(* Logix 5000 project; controller cal1615 1756-L62 rev 20.19; software revision 20.05; part 12 of 82 *)
(* tags used below, declared in another part *)
   tmrFlash : TIMER[4];   // Flash Timer
   aaa_aaa_temp : BOOL;
   FAULT : BOOL;   // Fault AFI
   FlashBit_500MSec : BOOL;   // Flash Bit 500 MSec
   HMI : BOOL;   // AFI HMI
   p00_FlashBit_1Sec : BOOL;   // System Flash Bit 1 Second
   p00_wac : Accumulator;   // Winder Accumulator
   p01_int_from_oxidizer : INT[10];   // System Oxidizer Int from Oxidizer
   p01_param_master_accel : REAL;   // Machine Parameter Master Accel Rate
   p01_param_master_decel : REAL;   // Machine Parameter Master Decel Rate
   p01_param_master_jog_accel : REAL;   // Machine Parameter Master Jog Acceleration mmpm/s
   p01_param_master_jog_decel : REAL;   // Machine Parameter Master Jog Deceleration mmpm/s
   p01_param_master_jog_speed : REAL;   // Machine Parameter Master Jog Speed
   p01_param_oven_timer_presets : DINT[32];   // System Parameter Oven Timer Presets
   p01_param_slow_speed_sp : REAL;   // System Parameters Slow Speed Setpoint
   p01_param_start_delay : REAL;   // Machine Parameter Start Delay
   p01_recipe_active : recipe;   // Active Recipe
   p01r01 : routine;
   p01r02_do_buzzer : BOOL;   // System Outputs Buzzer
   p01r02_do_horn : BOOL;   // System Outputs Horn
   p01r02_do_red_stack_light : BOOL;   // System Outputs Red Stack Light
   p01r02_do_yellow_stack_light : BOOL;   // System Outputs Yellow Stack Light
   p01r02_plc_scan_time_in_sec : REAL;   // System PLC Scan Time in Seconds
   p01r02_timer_second : TIMER[2];   // System Misc Control Timer Second Pulse
   p01r09 : routine;   // System Modes
   p01r09_mode_run : BOOL;   // System Modes All Modes Run Mode
   p01r09_open_oven : BOOL;
   p01r09_pb_global_reset : BOOL;   // System Modes PB: Global Fault Reset
   p01r09_pb_line_jog : BOOL;   // System Modes PB: Line Jog Forward
   p01r09_request_line_jog : BOOL;   // System Modes Request Line Jog Forward
   p01r10 : routine;   // System Annunciators
   p01r10_timer_fault : TIMER[4];   // System Fault Delay
   p01r10_timer_warning : TIMER[4];   // System Warning Delay
   p01r11 : routine;   // System Timer Presets
   p01r11_timer_fault : TIMER[4];   // System Fault Delay
   p01r11_timer_warning : TIMER[4];   // System Warning Delay
   p01r12 : routine;   // System Line Accel Decel Control
   p01r12_accel_rate : REAL;   // Machine Parameter Master Jog Acceleration mmpm/s
   p01r12_decel_rate : REAL;   // Machine Parameter Master Jog Deceleration mmpm/s
   p01r12_line_at_speed : BOOL;
   p01r12_master_acel_decel_ramp : SYS_ACC_DEC_RAMP;   // System Line Accel Decel Control Ramp
   p01r12_master_ramped_speed : REAL;   // System Line Accel Decel Control Master Ramped Speed
   p01r12_ramped_setpoint : REAL;   // System Line Accel Decel Control Ramped Setpoint
   p01r12_request_any_jog_thread : BOOL;   // System Line Accel Decel Control Request Any Jog/Thread
   p01r12_selected_line_speed : REAL;   // System Line Accel Decel Control Selected Line Speed
   p01r12_timer_fault : TIMER[8];   // System Line Start Sequence Fault Delay
   p01r12_timer_warning : TIMER[8];   // System Line Start Sequence Warning Delay
   p01r12_zero_line_speed : BOOL;   // System Line Accel Decel Control Line Speed at Zero
   p01r13 : routine;   // System Line Start Sequence
   p01r13_LFL_stop : BOOL;   // System Line Stop from LFL
   p01r13_line_running : BOOL;   // System Line Start Sequence Line Running
   p01r13_line_slow_ramp : BOOL;   // System Line Start Sequence Start Line to Slow Speed
   p01r13_oven_temp_ok : BOOL;   // System Line Start Sequence Oven Temperature Ready
   p01r13_pb_start : BOOL;   // System Line Start Sequence PB: Line Start
   p01r13_pb_stop : BOOL;   // System Line Start Sequence PB: Line Stop
   p01r13_permissive_drives : BOOL;   // System Line Start Sequence Permissive Drives
   p01r13_permissive_line_run : BOOL;   // System Line Start Sequence Permissive Line Run
   p01r13_permissive_oven : BOOL;   // System Line start Sequence Permissive Ovens
   p01r13_permissive_oxidizer : BOOL;   // System Line Start Sequence Permissive Oxidizer
   p01r13_request_run : BOOL;   // System Line Start Sequence Request Run
   p01r13_request_stop : BOOL;   // System Line Start Sequence Request Stop
   p01r13_state : DINT;   // System Line Start Sequence Sequencer Step
   p01r13_system_mode_run : BOOL;   // System Line Start Sequence All Drive Sections in Run Mode
   p01r13_temperature_status_check : TIMER;   // System Line Start Sequence Temperature Check
   p01r13_timer_line_start_warning_dwell : TIMER;   // System Line Start Sequence Pre Start Warning Dwell Timer
   p01r14 : routine;
   p02_dint_from_hmi : hmi_dint;
   p02_real_from_hmi : hmi_real;   // MOP HMI Iface Real from HMI
   p11r30 : routine;   // Zone 1 Temperature Control
   p11r30_request_heat : BOOL;   // Zone 1 Temperature Control Request Heat
   p11r31 : routine;   // Zone 1 Exhaust VFD
   p12r30 : routine;   // Zone 2 Temperature Control
   p12r30_request_heat : BOOL;   // Zone 2 Temperature Control Request Heat
   p12r31 : routine;   // Zone 2 Exhaust VFD
   p13r30 : routine;   // Zone 3 Temperature Control
   p13r30_request_cool : BOOL;   // Zone 3 Temperature Control Request Cooling
   p20_do_close_nip : BOOL;   // Letoff Digital Output Feedroll Roll Nip Close
   p20r02_letoff_selection_dwell : TIMER;
   p20r10 : routine;   // Letoff Letoff Tension Control
   p20r15 : routine;   // Letoff Letoff A VFD
   p20r15_loa_on : BOOL;   // Letoff Letoff A VFD On
   p20r16 : routine;   // Letoff Letoff B VFD
   p20r16_lob_on : BOOL;   // Letoff Letoff B On
   p20r18_index_complete : BOOL;   // Letoff Letoff Turret VFD Index Complete
   p22_param_ts1_jog_speed : REAL;   // System Parameter Tension Stand 1 Jog Speed
   p22r09_mode_run : BOOL;   // Tension Stand 1 Modes Run Mode
   p22r09_mode_thread : BOOL;   // Tension Stand 1 Modes Thread Mode
   p22r09_pb_jog_fwd : BOOL;   // Tension Stand 1 Modes PB: Jog Forward
   p22r09_pb_jog_rev : BOOL;   // Tension Stand 1 Modes PB: Jog Reverse
   p22r11 : routine;   // Tension Stand 1 VFD
   p22r11_request_thread_fwd : BOOL;   // Tension Stand 1 VFD Request Thread FWD
   p22r11_request_thread_rev : BOOL;   // Tension Stand 1 VFD Request Thread REV
   p23_di_impreg_tank_up : BOOL;   // Input Impreg Dip Tank Up
   p23_param_mtr_jog_speed : REAL;   // System Parameter Metering Roll Jog Speed
   p23r02 : routine;   // Impreg Misc Control
   p23r15 : routine;   // Impreg Metering Roll VFD
   p25_param_ts2_jog_speed : REAL;   // System Parameter Tension Stand 2 Jog Speed
   p25r09_mode_run : BOOL;   // Tension Stand 2 Modes Run Mode
   p25r09_mode_thread : BOOL;   // Tension Stand 2 Modes Thread Mode
   p25r09_pb_jog_fwd : BOOL;   // Tension Stand 2 Modes PB: Jog Forward
   p25r09_pb_jog_rev : BOOL;   // Tension Stand 2 Modes PB: Jog Reverse
   p25r11 : routine;   // Tension Stand 2 VFD
   p25r11_request_thread_fwd : BOOL;   // Tension Stand 2 VFD Request Thread FWD
   p25r11_request_thread_rev : BOOL;   // Tension Stand 2 VFD Request Thread REV
   p28r11 : routine;
   p29_param_winder_jog_speed : REAL;   // System Parameters Winder Jog Speed
   p29r11_line_start : BOOL;
   p29r11_line_stop : BOOL;
   p29r15 : routine;   // Winder Winder A VFD
   p29r16 : routine;   // Winder Winder B VFD
   p31r09 : routine;   // Edge Control Modes
(* P01_System, continued *)

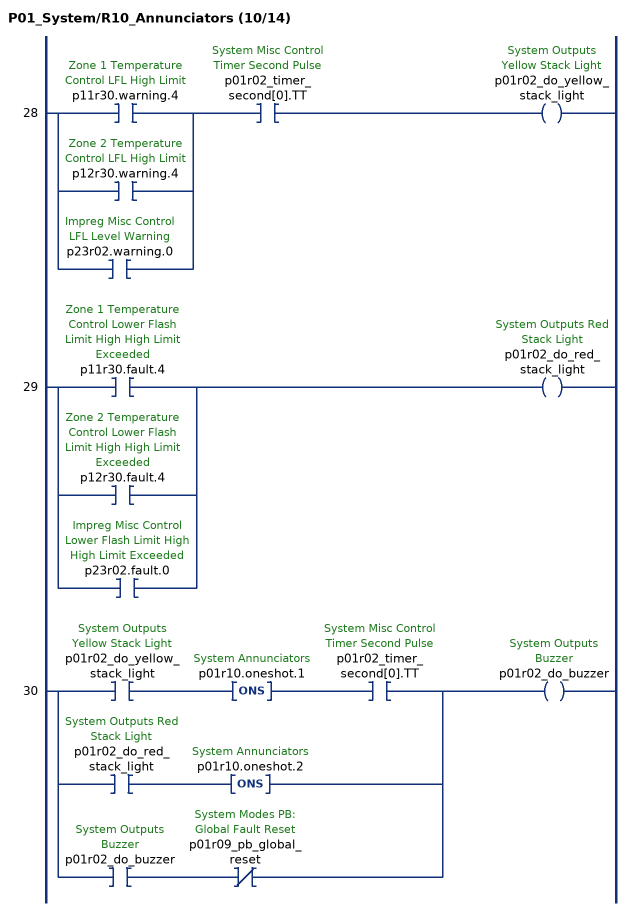
   [picture p138: P01_System/R10_Annunciators rungs 28-30]
   28: [XIC(p11r30.warning.4) ,XIC(p12r30.warning.4) ,XIC(p23r02.warning.0) ]XIC(p01r02_timer_second[0].TT)OTE(p01r02_do_yellow_stack_light);
   29: [XIC(p11r30.fault.4) ,XIC(p12r30.fault.4) ,XIC(p23r02.fault.0) ]OTE(p01r02_do_red_stack_light);
   30: [[XIC(p01r02_do_yellow_stack_light) ONS(p01r10.oneshot.1) XIC(p01r02_timer_second[0].TT) ,XIC(p01r02_do_red_stack_light) ONS(p01r10.oneshot.2) ] ,XIC(p01r02_do_buzzer) XIO(p01r09_pb_global_reset) ]OTE(p01r02_do_buzzer);
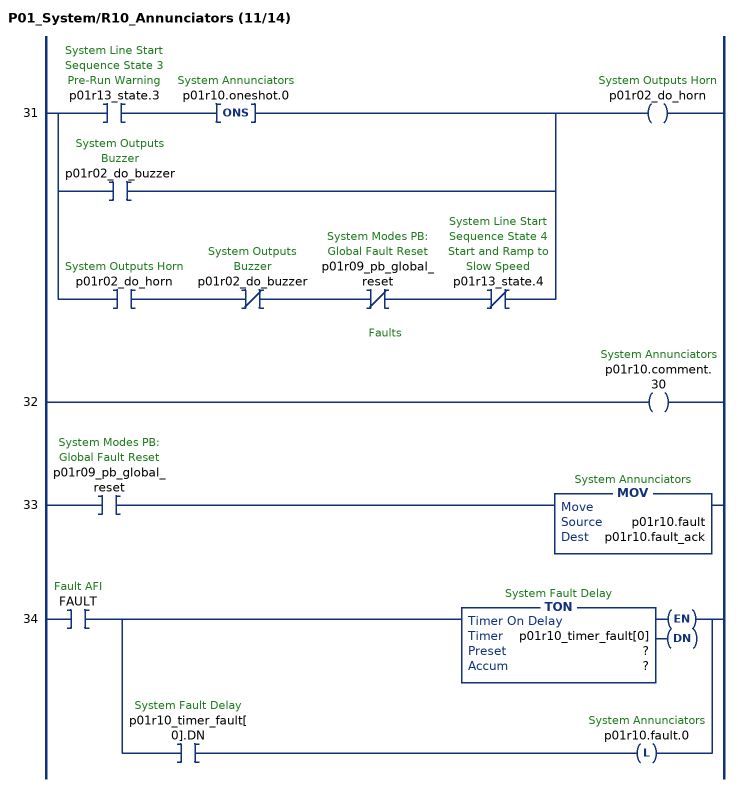
   31: [[XIC(p01r13_state.3) ONS(p01r10.oneshot.0) ,XIC(p01r02_do_buzzer) ] ,XIC(p01r02_do_horn) XIO(p01r02_do_buzzer) XIO(p01r09_pb_global_reset) XIO(p01r13_state.4) ]OTE(p01r02_do_horn);
   // Faults
   32: OTE(p01r10.comment.30);
   33: XIC(p01r09_pb_global_reset)MOV(p01r10.fault,p01r10.fault_ack);
   34: XIC(FAULT)[TON(p01r10_timer_fault[0],?,?) ,XIC(p01r10_timer_fault[0].DN) OTL(p01r10.fault.0) ];
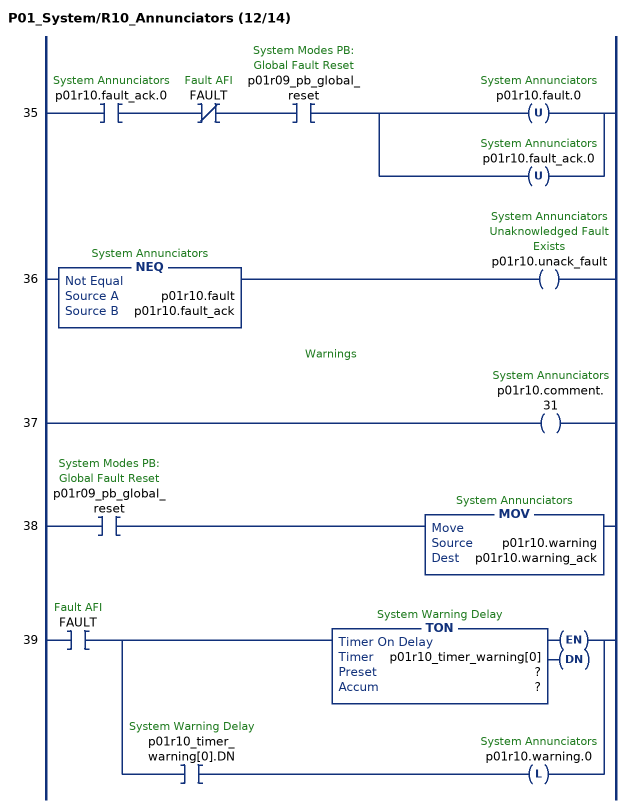
   35: XIC(p01r10.fault_ack.0)XIO(FAULT)XIC(p01r09_pb_global_reset)[OTU(p01r10.fault.0) ,OTU(p01r10.fault_ack.0) ];
   36: NEQ(p01r10.fault,p01r10.fault_ack)OTE(p01r10.unack_fault);
   // Warnings
   37: OTE(p01r10.comment.31);
   38: XIC(p01r09_pb_global_reset)MOV(p01r10.warning,p01r10.warning_ack);
   39: XIC(FAULT)[TON(p01r10_timer_warning[0],?,?) ,XIC(p01r10_timer_warning[0].DN) OTL(p01r10.warning.0) ];
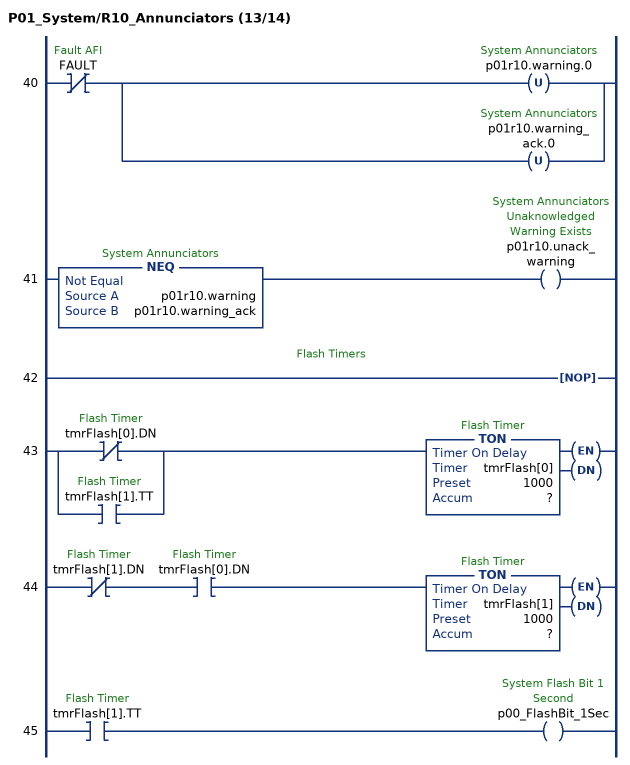
   40: XIO(FAULT)[OTU(p01r10.warning.0) ,OTU(p01r10.warning_ack.0) ];
   41: NEQ(p01r10.warning,p01r10.warning_ack)OTE(p01r10.unack_warning);
   // Flash Timers
   42: NOP();
   43: [XIO(tmrFlash[0].DN) ,XIC(tmrFlash[1].TT) ]TON(tmrFlash[0],?,?);
   44: XIO(tmrFlash[1].DN)XIC(tmrFlash[0].DN)TON(tmrFlash[1],?,?);
   45: XIC(tmrFlash[1].TT)OTE(p00_FlashBit_1Sec);
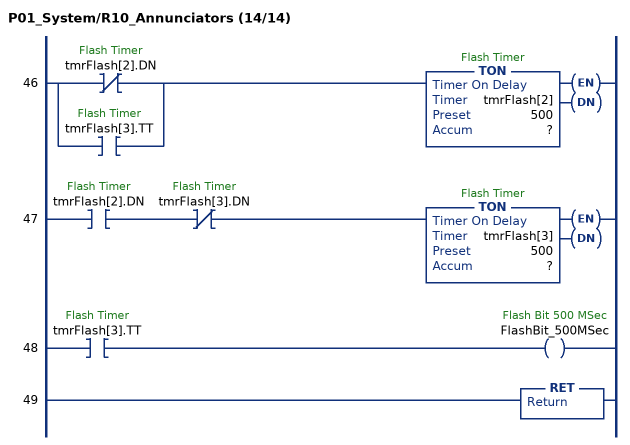
   46: [XIO(tmrFlash[2].DN) ,XIC(tmrFlash[3].TT) ]TON(tmrFlash[2],?,?);
   47: XIC(tmrFlash[2].DN)XIO(tmrFlash[3].DN)TON(tmrFlash[3],?,?);
   48: XIC(tmrFlash[3].TT)OTE(FlashBit_500MSec);
   49: RET();
END_ROUTINE

ROUTINE R11_Oven_Timer_Presets   (* ladder *)
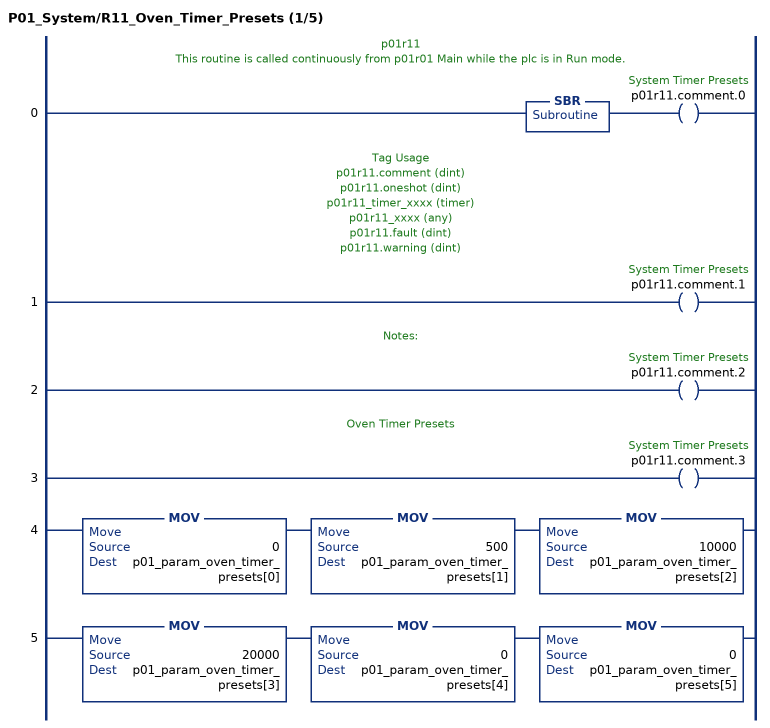
   // p01r11
   // This routine is called continuously from p01r01 Main while the plc is in Run mode.
   0: SBR()OTE(p01r11.comment.0);
   // Tag Usage
   // p01r11.comment (dint)
   // p01r11.oneshot (dint)
   // p01r11_timer_xxxx (timer)
   // p01r11_xxxx (any)
   // p01r11.fault (dint)
   // p01r11.warning (dint)
   1: OTE(p01r11.comment.1);
   // Notes:
   2: OTE(p01r11.comment.2);
   // Oven Timer Presets
   3: OTE(p01r11.comment.3);
   4: MOV(0,p01_param_oven_timer_presets[0])MOV(500,p01_param_oven_timer_presets[1])MOV(10000,p01_param_oven_timer_presets[2]);
   5: MOV(20000,p01_param_oven_timer_presets[3])MOV(0,p01_param_oven_timer_presets[4])MOV(0,p01_param_oven_timer_presets[5]);
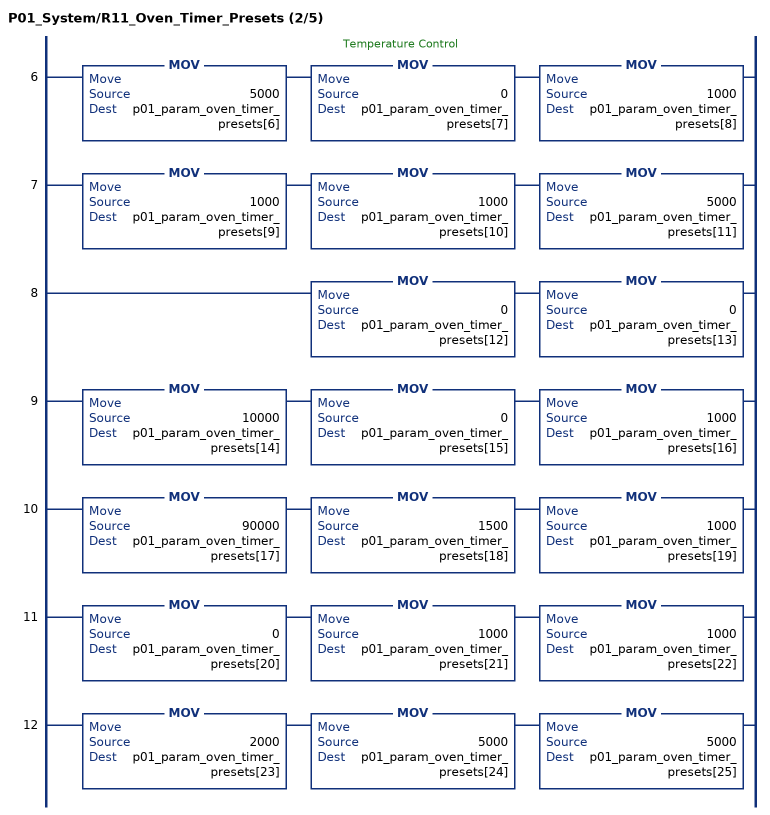
   // Temperature Control
   6: MOV(5000,p01_param_oven_timer_presets[6])MOV(0,p01_param_oven_timer_presets[7])MOV(1000,p01_param_oven_timer_presets[8]);
   7: MOV(1000,p01_param_oven_timer_presets[9])MOV(1000,p01_param_oven_timer_presets[10])MOV(5000,p01_param_oven_timer_presets[11]);
   8: MOV(0,p01_param_oven_timer_presets[12])MOV(0,p01_param_oven_timer_presets[13]);
   9: MOV(10000,p01_param_oven_timer_presets[14])MOV(0,p01_param_oven_timer_presets[15])MOV(1000,p01_param_oven_timer_presets[16]);
   10: MOV(90000,p01_param_oven_timer_presets[17])MOV(1500,p01_param_oven_timer_presets[18])MOV(1000,p01_param_oven_timer_presets[19]);
   11: MOV(0,p01_param_oven_timer_presets[20])MOV(1000,p01_param_oven_timer_presets[21])MOV(1000,p01_param_oven_timer_presets[22]);
   12: MOV(2000,p01_param_oven_timer_presets[23])MOV(5000,p01_param_oven_timer_presets[24])MOV(5000,p01_param_oven_timer_presets[25]);
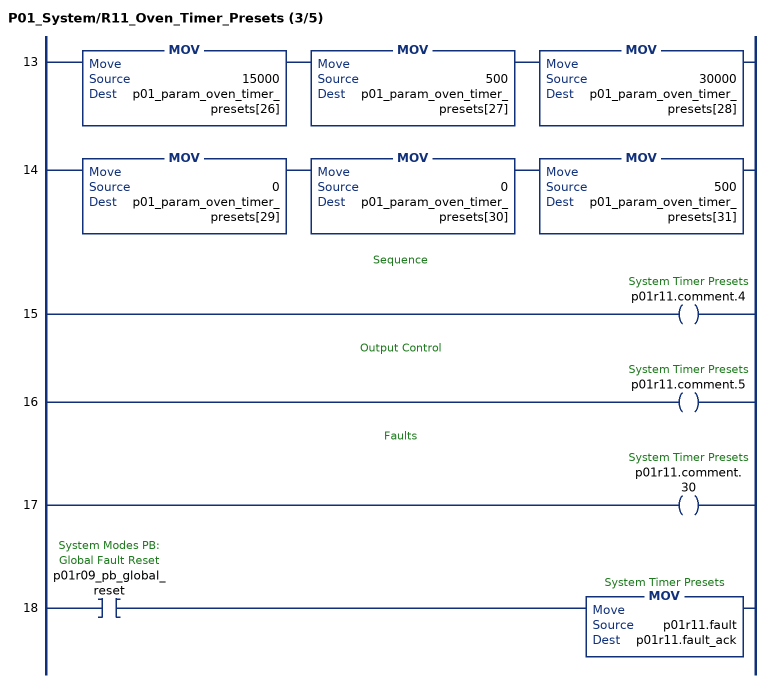
   13: MOV(15000,p01_param_oven_timer_presets[26])MOV(500,p01_param_oven_timer_presets[27])MOV(30000,p01_param_oven_timer_presets[28]);
   14: MOV(0,p01_param_oven_timer_presets[29])MOV(0,p01_param_oven_timer_presets[30])MOV(500,p01_param_oven_timer_presets[31]);
   // Sequence
   15: OTE(p01r11.comment.4);
   // Output Control
   16: OTE(p01r11.comment.5);
   // Faults
   17: OTE(p01r11.comment.30);
   18: XIC(p01r09_pb_global_reset)MOV(p01r11.fault,p01r11.fault_ack);
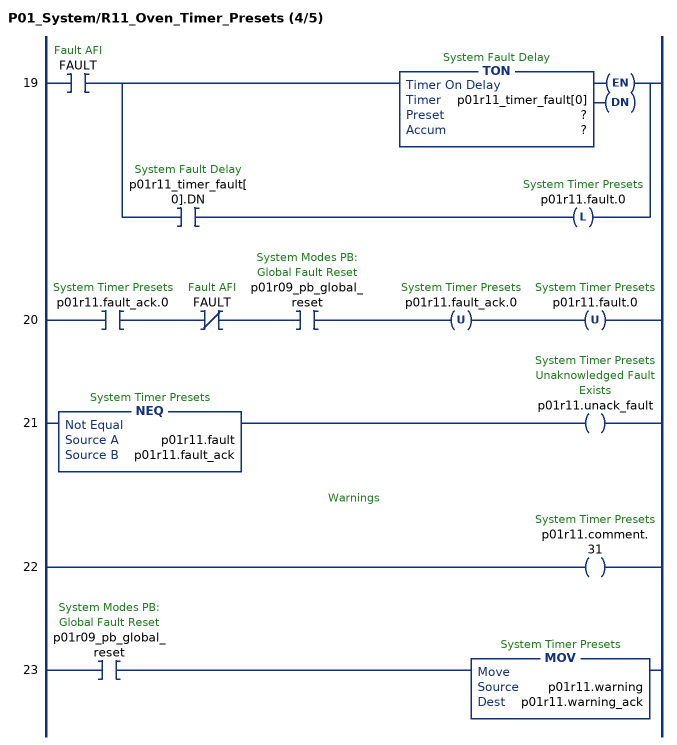
   19: XIC(FAULT)[TON(p01r11_timer_fault[0],?,?) ,XIC(p01r11_timer_fault[0].DN) OTL(p01r11.fault.0) ];
   20: XIC(p01r11.fault_ack.0)XIO(FAULT)XIC(p01r09_pb_global_reset)OTU(p01r11.fault_ack.0)OTU(p01r11.fault.0);
   21: NEQ(p01r11.fault,p01r11.fault_ack)OTE(p01r11.unack_fault);
   // Warnings
   22: OTE(p01r11.comment.31);
   23: XIC(p01r09_pb_global_reset)MOV(p01r11.warning,p01r11.warning_ack);
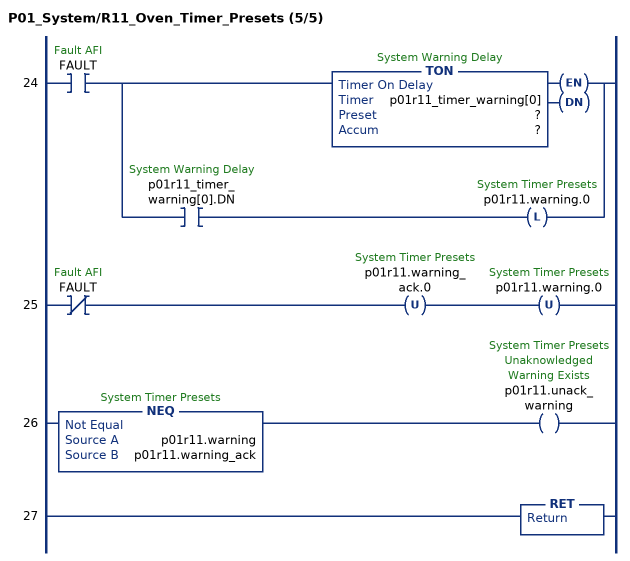
   24: XIC(FAULT)[TON(p01r11_timer_warning[0],?,?) ,XIC(p01r11_timer_warning[0].DN) OTL(p01r11.warning.0) ];
   25: XIO(FAULT)OTU(p01r11.warning_ack.0)OTU(p01r11.warning.0);
   26: NEQ(p01r11.warning,p01r11.warning_ack)OTE(p01r11.unack_warning);
   27: RET();
END_ROUTINE

ROUTINE R12_Line_Accel_Decel_Control   (* ladder *)
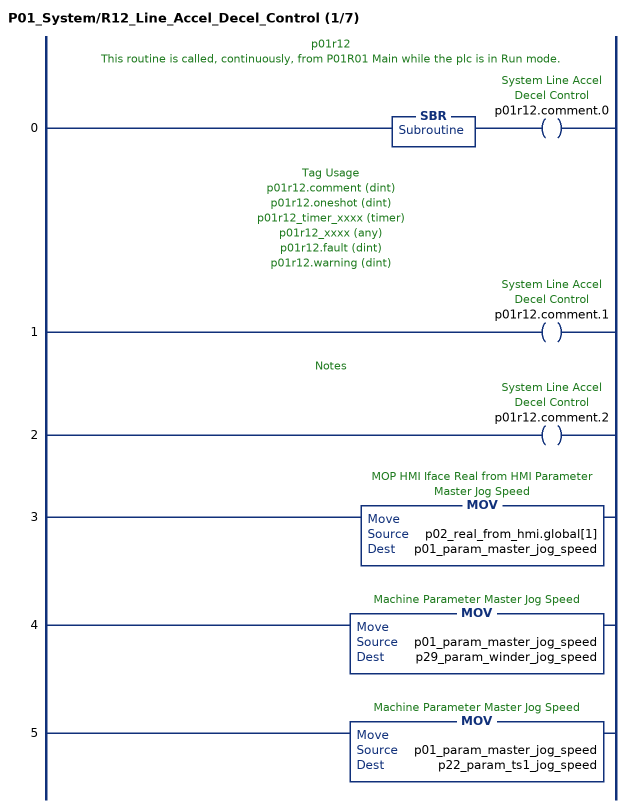
   // p01r12
   // This routine is called, continuously, from P01R01 Main while the plc is in Run mode.
   0: SBR()OTE(p01r12.comment.0);
   // Tag Usage
   // p01r12.comment (dint)
   // p01r12.oneshot (dint)
   // p01r12_timer_xxxx (timer)
   // p01r12_xxxx (any)
   // p01r12.fault (dint)
   // p01r12.warning (dint)
   1: OTE(p01r12.comment.1);
   // Notes
   2: OTE(p01r12.comment.2);
   3: MOV(p02_real_from_hmi.global[1],p01_param_master_jog_speed);
   4: MOV(p01_param_master_jog_speed,p29_param_winder_jog_speed);
   5: MOV(p01_param_master_jog_speed,p22_param_ts1_jog_speed);
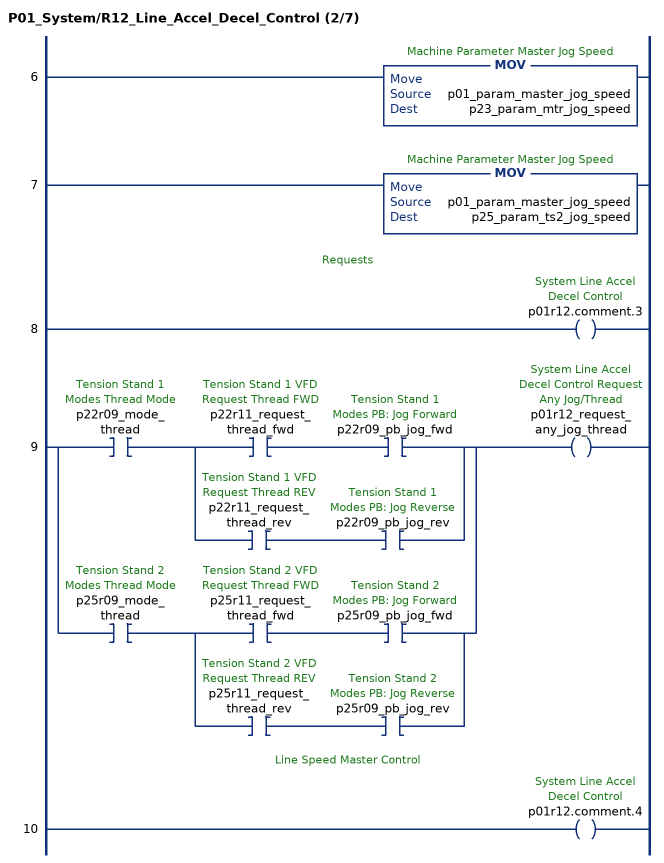
   6: MOV(p01_param_master_jog_speed,p23_param_mtr_jog_speed);
   7: MOV(p01_param_master_jog_speed,p25_param_ts2_jog_speed);
   // Requests
   8: OTE(p01r12.comment.3);
   9: [XIC(p22r09_mode_thread) [XIC(p22r11_request_thread_fwd) XIC(p22r09_pb_jog_fwd) ,XIC(p22r11_request_thread_rev) XIC(p22r09_pb_jog_rev) ] ,XIC(p25r09_mode_thread) [XIC(p25r11_request_thread_fwd) XIC(p25r09_pb_jog_fwd) ,XIC(p25r11_request_thread_rev) XIC(p25r09_pb_jog_rev) ] ]OTE(p01r12_request_any_jog_thread);
   // Line Speed Master Control
   10: OTE(p01r12.comment.4);
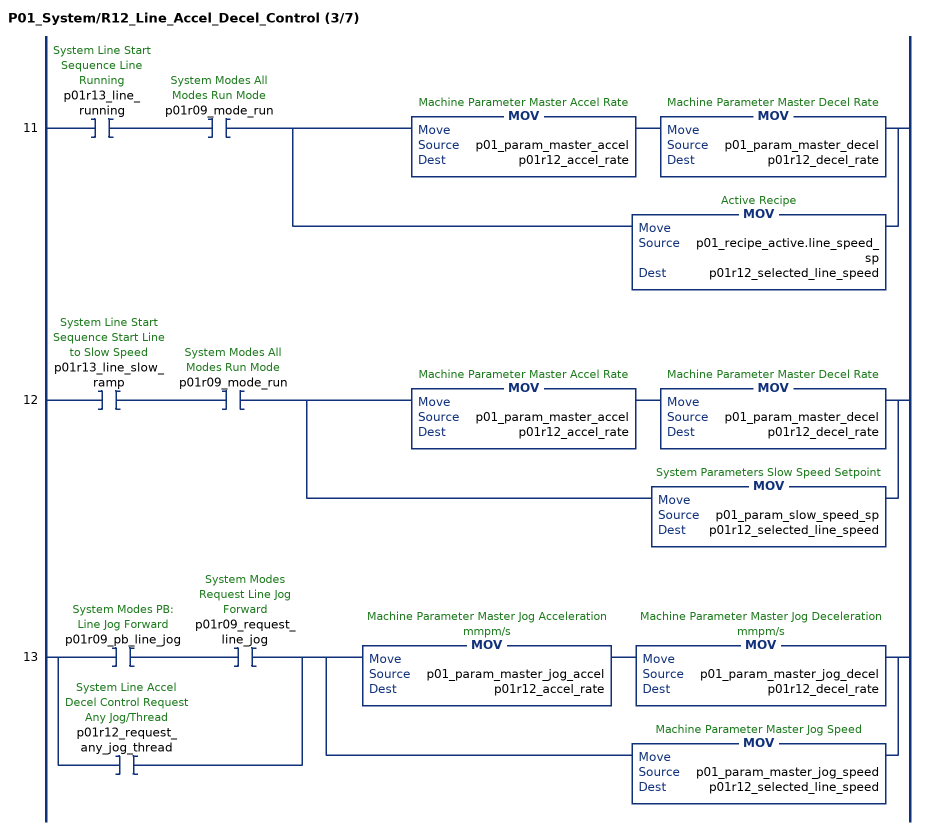
   11: XIC(p01r13_line_running)XIC(p01r09_mode_run)[MOV(p01_param_master_accel,p01r12_accel_rate) MOV(p01_param_master_decel,p01r12_decel_rate) ,MOV(p01_recipe_active.line_speed_sp,p01r12_selected_line_speed) ];
   12: XIC(p01r13_line_slow_ramp)XIC(p01r09_mode_run)[MOV(p01_param_master_accel,p01r12_accel_rate) MOV(p01_param_master_decel,p01r12_decel_rate) ,MOV(p01_param_slow_speed_sp,p01r12_selected_line_speed) ];
   13: [XIC(p01r09_pb_line_jog) XIC(p01r09_request_line_jog) ,XIC(p01r12_request_any_jog_thread) ][MOV(p01_param_master_jog_accel,p01r12_accel_rate) MOV(p01_param_master_jog_decel,p01r12_decel_rate) ,MOV(p01_param_master_jog_speed,p01r12_selected_line_speed) ];
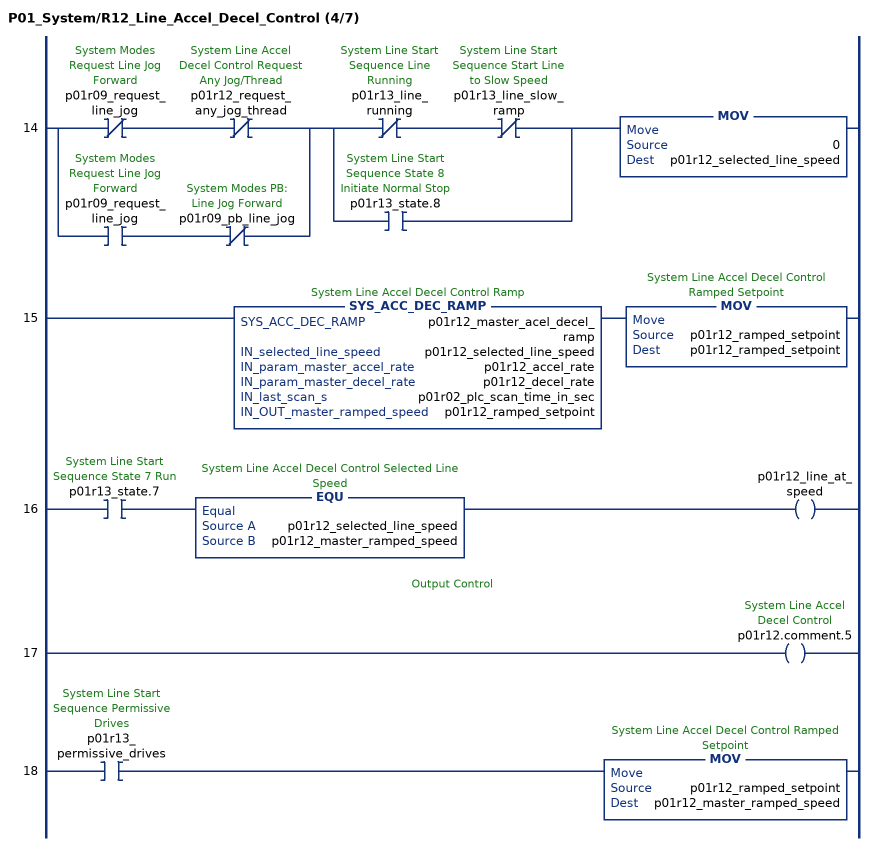
   14: [XIO(p01r09_request_line_jog) XIO(p01r12_request_any_jog_thread) ,XIC(p01r09_request_line_jog) XIO(p01r09_pb_line_jog) ][XIO(p01r13_line_running) XIO(p01r13_line_slow_ramp) ,XIC(p01r13_state.8) ]MOV(0,p01r12_selected_line_speed);
   15: SYS_ACC_DEC_RAMP(p01r12_master_acel_decel_ramp,p01r12_selected_line_speed,p01r12_accel_rate,p01r12_decel_rate,p01r02_plc_scan_time_in_sec,p01r12_ramped_setpoint)MOV(p01r12_ramped_setpoint,p01r12_ramped_setpoint);
   16: XIC(p01r13_state.7)EQU(p01r12_selected_line_speed,p01r12_master_ramped_speed)OTE(p01r12_line_at_speed);
   // Output Control
   17: OTE(p01r12.comment.5);
   18: XIC(p01r13_permissive_drives)MOV(p01r12_ramped_setpoint,p01r12_master_ramped_speed);
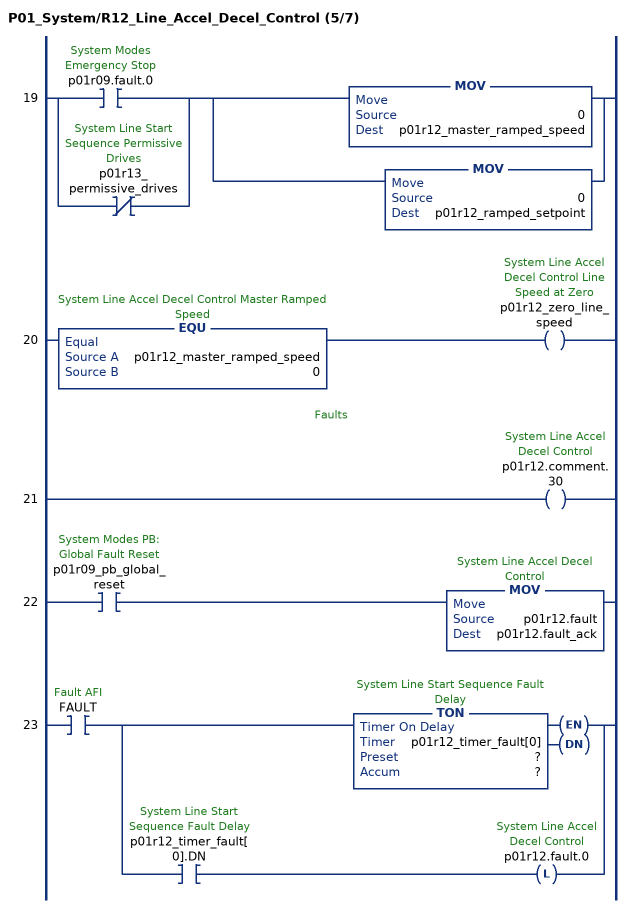
   19: [XIC(p01r09.fault.0) ,XIO(p01r13_permissive_drives) ][MOV(0,p01r12_master_ramped_speed) ,MOV(0,p01r12_ramped_setpoint) ];
   20: EQU(p01r12_master_ramped_speed,0)OTE(p01r12_zero_line_speed);
   // Faults
   21: OTE(p01r12.comment.30);
   22: XIC(p01r09_pb_global_reset)MOV(p01r12.fault,p01r12.fault_ack);
   23: XIC(FAULT)[TON(p01r12_timer_fault[0],?,?) ,XIC(p01r12_timer_fault[0].DN) OTL(p01r12.fault.0) ];
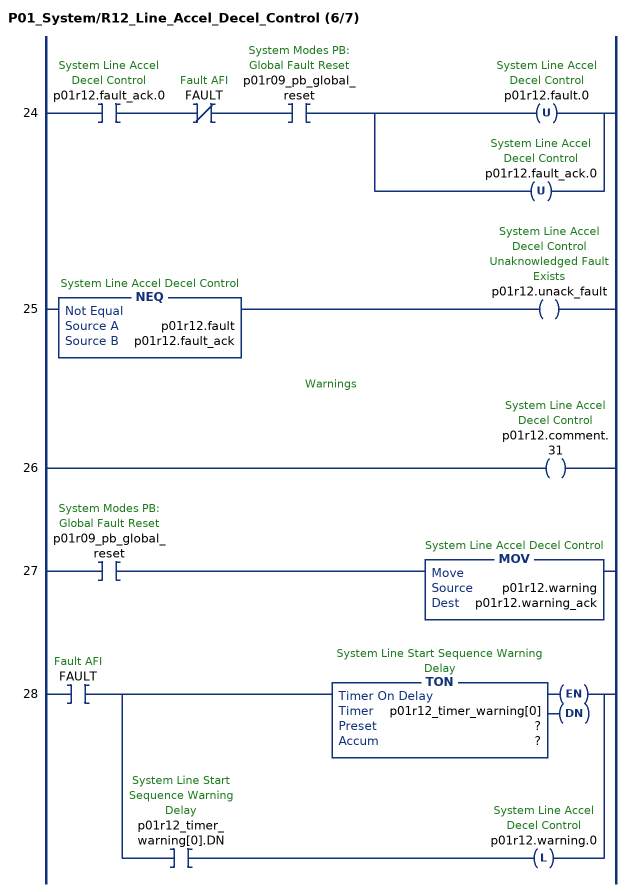
   24: XIC(p01r12.fault_ack.0)XIO(FAULT)XIC(p01r09_pb_global_reset)[OTU(p01r12.fault.0) ,OTU(p01r12.fault_ack.0) ];
   25: NEQ(p01r12.fault,p01r12.fault_ack)OTE(p01r12.unack_fault);
   // Warnings
   26: OTE(p01r12.comment.31);
   27: XIC(p01r09_pb_global_reset)MOV(p01r12.warning,p01r12.warning_ack);
   28: XIC(FAULT)[TON(p01r12_timer_warning[0],?,?) ,XIC(p01r12_timer_warning[0].DN) OTL(p01r12.warning.0) ];
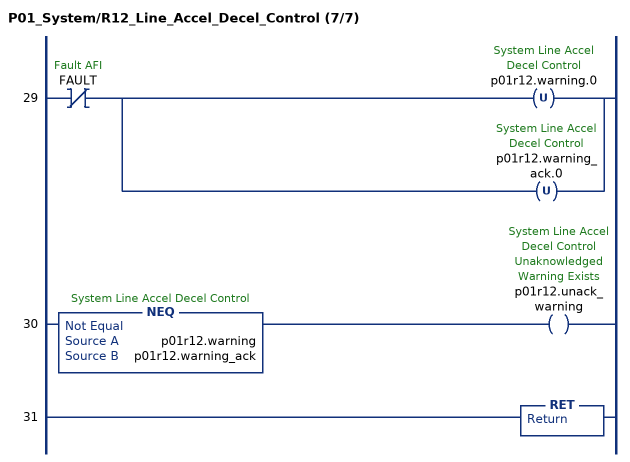
   29: XIO(FAULT)[OTU(p01r12.warning.0) ,OTU(p01r12.warning_ack.0) ];
   30: NEQ(p01r12.warning,p01r12.warning_ack)OTE(p01r12.unack_warning);
   31: RET();
END_ROUTINE

ROUTINE R13_Line_Start_Sequence   (* ladder *)
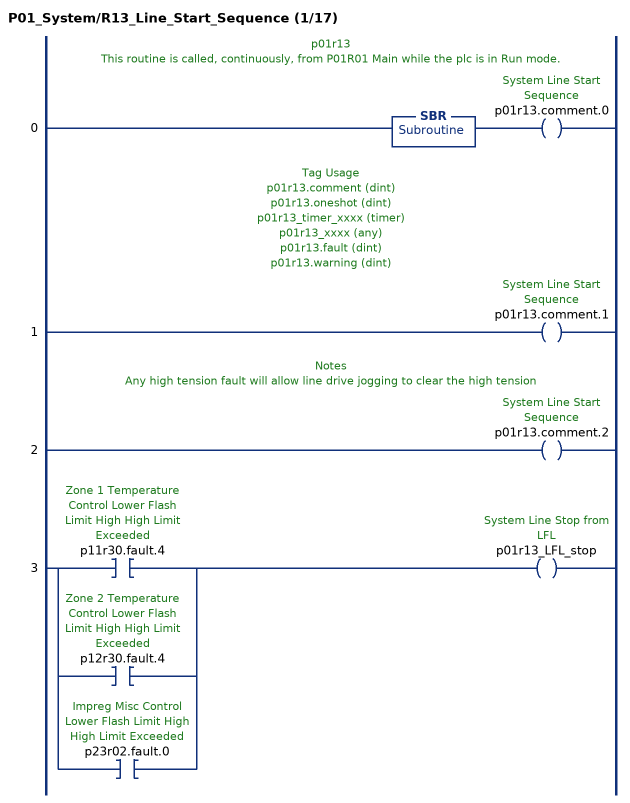
   // p01r13
   // This routine is called, continuously, from P01R01 Main while the plc is in Run mode.
   0: SBR()OTE(p01r13.comment.0);
   // Tag Usage
   // p01r13.comment (dint)
   // p01r13.oneshot (dint)
   // p01r13_timer_xxxx (timer)
   // p01r13_xxxx (any)
   // p01r13.fault (dint)
   // p01r13.warning (dint)
   1: OTE(p01r13.comment.1);
   // Notes
   // Any high tension fault will allow line drive jogging to clear the high tension
   2: OTE(p01r13.comment.2);
   3: [XIC(p11r30.fault.4) ,XIC(p12r30.fault.4) ,XIC(p23r02.fault.0) ]OTE(p01r13_LFL_stop);
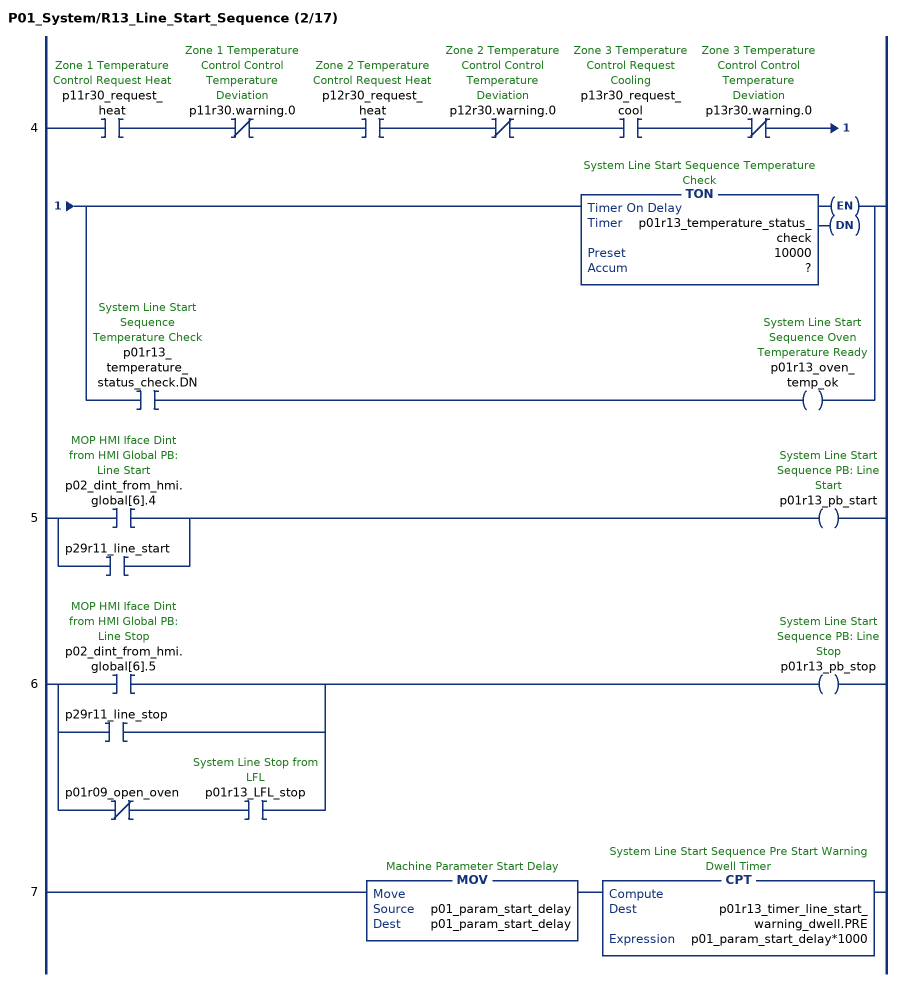
   4: XIC(p11r30_request_heat)XIO(p11r30.warning.0)XIC(p12r30_request_heat)XIO(p12r30.warning.0)XIC(p13r30_request_cool)XIO(p13r30.warning.0)[TON(p01r13_temperature_status_check,?,?) ,XIC(p01r13_temperature_status_check.DN) OTE(p01r13_oven_temp_ok) ];
   5: [XIC(p02_dint_from_hmi.global[6].4) ,XIC(p29r11_line_start) ]OTE(p01r13_pb_start);
   6: [XIC(p02_dint_from_hmi.global[6].5) ,XIC(p29r11_line_stop) ,XIO(p01r09_open_oven) XIC(p01r13_LFL_stop) ]OTE(p01r13_pb_stop);
   7: MOV(p01_param_start_delay,p01_param_start_delay)CPT(p01r13_timer_line_start_warning_dwell.PRE,p01_param_start_delay*1000);
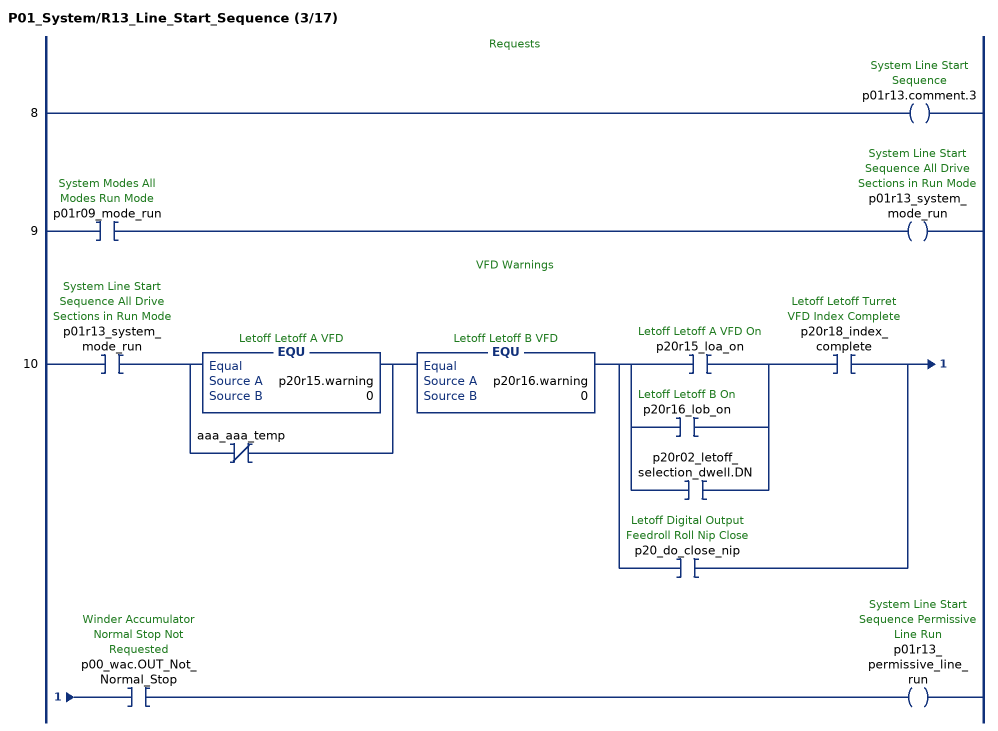
   // Requests
   8: OTE(p01r13.comment.3);
   9: XIC(p01r09_mode_run)OTE(p01r13_system_mode_run);
   // VFD Warnings
   10: XIC(p01r13_system_mode_run)[EQU(p20r15.warning,0) ,XIO(aaa_aaa_temp) ]EQU(p20r16.warning,0)[[XIC(p20r15_loa_on) ,XIC(p20r16_lob_on) ,XIC(p20r02_letoff_selection_dwell.DN) ] XIC(p20r18_index_complete) ,XIC(p20_do_close_nip) ]XIC(p00_wac.OUT_Not_Normal_Stop)OTE(p01r13_permissive_line_run);
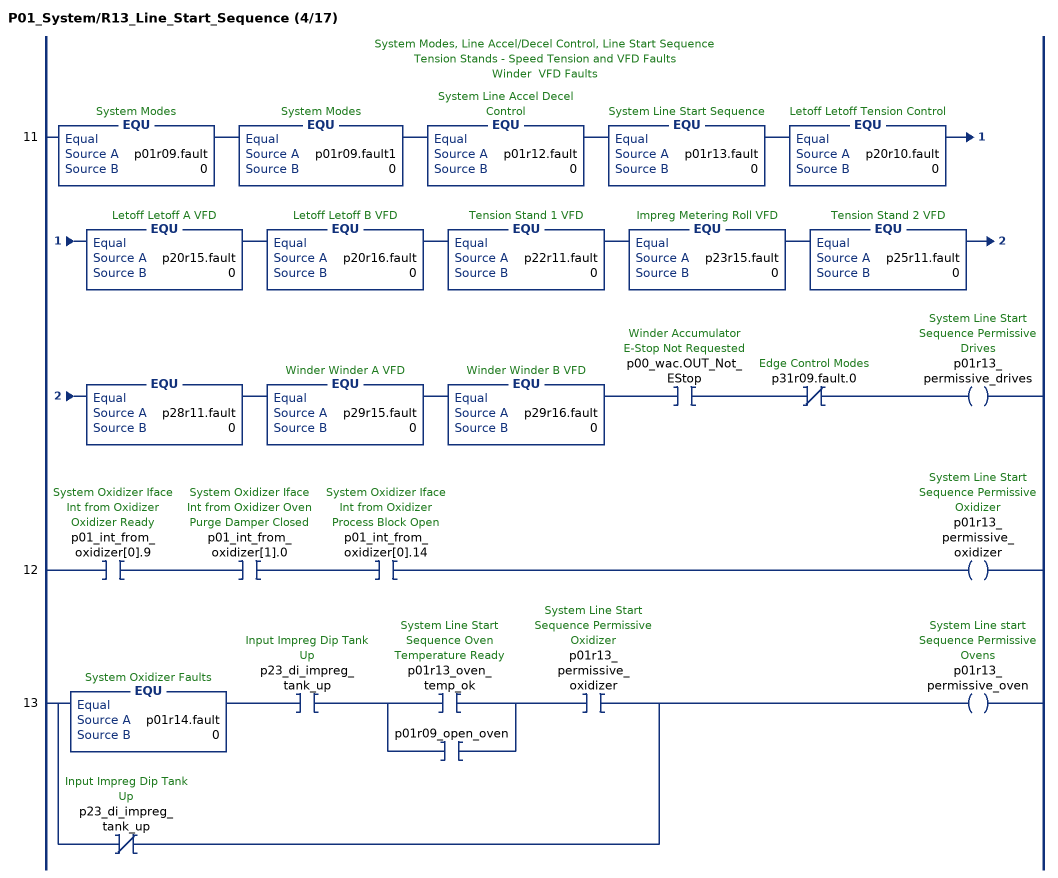
   // System Modes, Line Accel/Decel Control, Line Start Sequence
   // Tension Stands - Speed Tension and VFD Faults
   // Winder  VFD Faults
   11: EQU(p01r09.fault,0)EQU(p01r09.fault1,0)EQU(p01r12.fault,0)EQU(p01r13.fault,0)EQU(p20r10.fault,0)EQU(p20r15.fault,0)EQU(p20r16.fault,0)EQU(p22r11.fault,0)EQU(p23r15.fault,0)EQU(p25r11.fault,0)EQU(p28r11.fault,0)EQU(p29r15.fault,0)EQU(p29r16.fault,0)XIC(p00_wac.OUT_Not_EStop)XIO(p31r09.fault.0)OTE(p01r13_permissive_drives);
   12: XIC(p01_int_from_oxidizer[0].9)XIC(p01_int_from_oxidizer[1].0)XIC(p01_int_from_oxidizer[0].14)OTE(p01r13_permissive_oxidizer);
   13: [EQU(p01r14.fault,0) XIC(p23_di_impreg_tank_up) [XIC(p01r13_oven_temp_ok) ,XIC(p01r09_open_oven) ] XIC(p01r13_permissive_oxidizer) ,XIO(p23_di_impreg_tank_up) ]OTE(p01r13_permissive_oven);
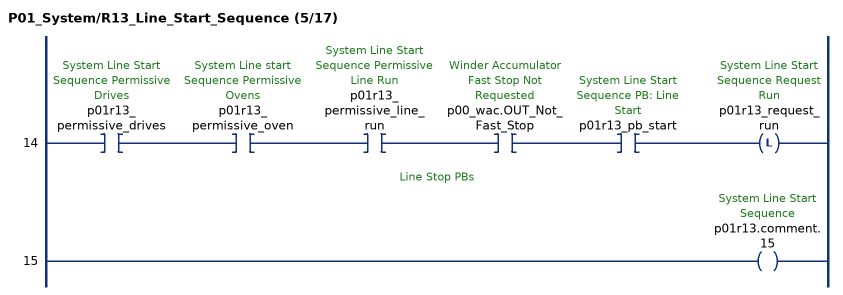
   14: XIC(p01r13_permissive_drives)XIC(p01r13_permissive_oven)XIC(p01r13_permissive_line_run)XIC(p00_wac.OUT_Not_Fast_Stop)XIC(p01r13_pb_start)OTL(p01r13_request_run);
   // Line Stop PBs
   15: OTE(p01r13.comment.15);
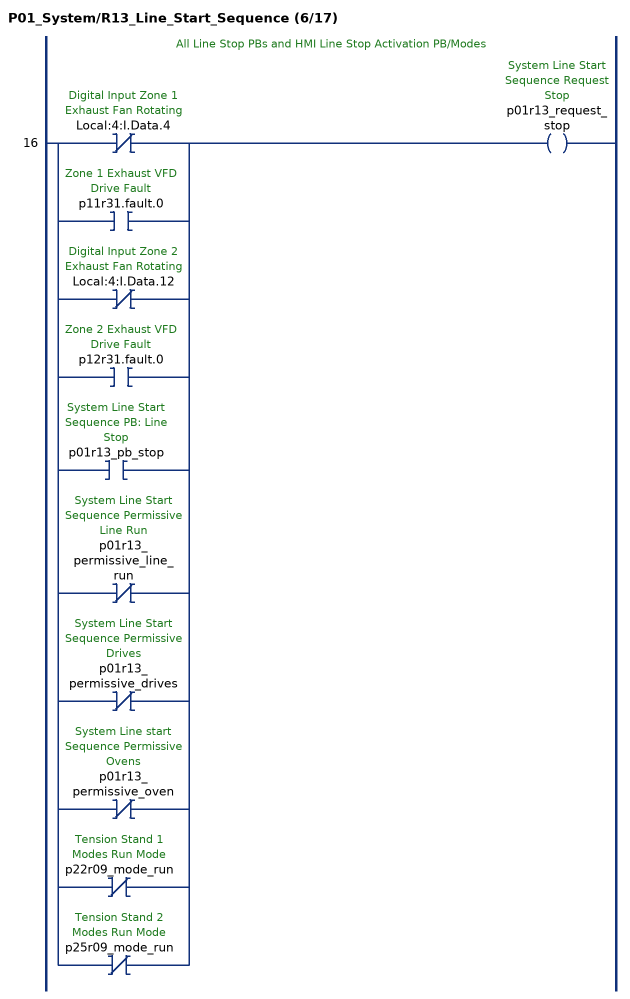
   // All Line Stop PBs and HMI Line Stop Activation PB/Modes
   16: [XIO(Local:4:I.Data.4) ,XIC(p11r31.fault.0) ,XIO(Local:4:I.Data.12) ,XIC(p12r31.fault.0) ,XIC(p01r13_pb_stop) ,XIO(p01r13_permissive_line_run) ,XIO(p01r13_permissive_drives) ,XIO(p01r13_permissive_oven) ,XIO(p22r09_mode_run) ,XIO(p25r09_mode_run) ]OTE(p01r13_request_stop);
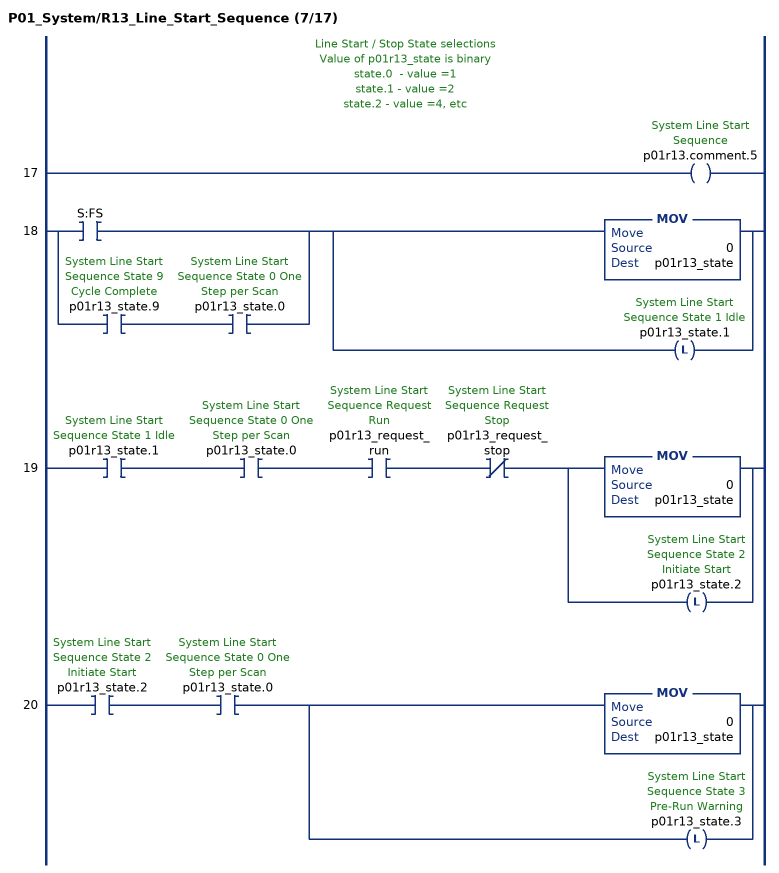
   // Line Start / Stop State selections
   // Value of p01r13_state is binary
   // state.0  - value =1
   // state.1 - value =2
   // state.2 - value =4, etc
   17: OTE(p01r13.comment.5);
   18: [XIC(S:FS) ,XIC(p01r13_state.9) XIC(p01r13_state.0) ][MOV(0,p01r13_state) ,OTL(p01r13_state.1) ];
   19: XIC(p01r13_state.1)XIC(p01r13_state.0)XIC(p01r13_request_run)XIO(p01r13_request_stop)[MOV(0,p01r13_state) ,OTL(p01r13_state.2) ];
   20: XIC(p01r13_state.2)XIC(p01r13_state.0)[MOV(0,p01r13_state) ,OTL(p01r13_state.3) ];
